FUNCTION_BLOCK SIMPLE_INIT (* Basic Function Block Type *)
  (* Standard: 61499-2 *)
  (* Version 0.0, 4/28/2023, Dmitrii, Flexbridge AB, Template *)
  PACKAGE UAO.Hackathon;
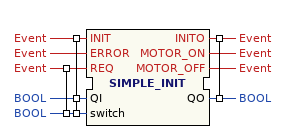
  EVENT_INPUT
    INIT WITH QI, switch; (* Initialization Request *)
    ERROR;
    REQ WITH switch;
  END_EVENT
  EVENT_OUTPUT
    INITO WITH QO; (* Initialization Confirm *)
    MOTOR_ON;
    MOTOR_OFF;
  END_EVENT
  VAR_INPUT
    QI : BOOL; (* Input event qualifier *)
    switch : BOOL;
  END_VAR
  VAR_OUTPUT
    QO : BOOL; (* Output event qualifier *)
  END_VAR
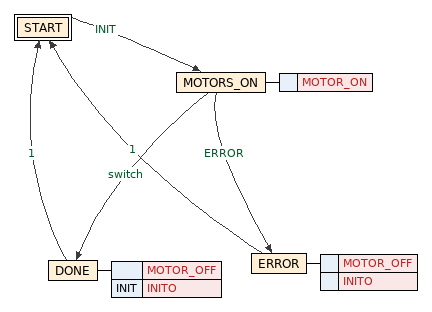
  EC_STATES
    START; (* Initial State *)
    MOTORS_ON : -> MOTOR_ON; (* Initialization *)
    DONE : -> MOTOR_OFF, INIT -> INITO;
    ERROR : -> MOTOR_OFF, -> INITO;
  END_STATES
  EC_TRANSITIONS
    START TO MOTORS_ON := INIT;
    MOTORS_ON TO ERROR := ERROR;
    MOTORS_ON TO DONE := switch;
    ERROR TO START := 1;
    DONE TO START := 1;
  END_TRANSITIONS
  ALGORITHM INIT IN ST: (* Initialization algorithm *)
QO:=TRUE;
  END_ALGORITHM
  ALGORITHM ERR IN ST:
QO:=FALSE;
  END_ALGORITHM
END_FUNCTION_BLOCK
